// TIA Portal V17 export
// export: Created 2024-08-07T21:44:12.0966309Z, ExportSetting WithDefaults, DisplayName Totally Integrated Automation Portal, DisplayVersion V17 Update 7, DisplayName TIA Portal Openness, DisplayVersion V17 Update 7, DisplayName TIA Portal Version Control Interface, DisplayVersion V17, DisplayName SINAMICS Startdrive Advanced, DisplayVersion V17 SP2, DisplayName SINAMICS Startdrive G110M, G120, G120C, G120D, G120P, G115D, DisplayVersion V17 SP2, DisplayName SINAMICS Startdrive G130, G150, S120, S150, SINAMICS MV, S210, DisplayVersion V17 SP2, DisplayName STEP 7 Professional, DisplayVersion V17 Update 7, DisplayName STEP 7 Safety, DisplayVersion V17 Update 6, DisplayName WinCC Advanced / Unified PC, DisplayVersion V17 Update 7
DATA_BLOCK "Default_SupervisionDB"   // DB68
VERSION : 0.1
// stored: AutoNumber true, DBAccessibleFromOPCUA true, DBAccessibleFromWebserver true, InstanceOfName Default_SupervisionFB, InstanceOfType FB
"Default_SupervisionFB"
   // VAR
   //    PC_Flags { ExternalWritable := 'False'; S7_SetPoint := 'True'} : PC_Flags_V2;
   //    State { ExternalWritable := 'False'; S7_SetPoint := 'True'} : SV_FB_State_V2;
   //    iOilHighLevekOK_O_1 { ExternalWritable := 'False'; S7_SetPoint := 'True'} : SV_State_V2;
   // END_VAR
BEGIN
END_DATA_BLOCK
